TEXTLIST tlStations
  200 = 'Loading Station' | EN: 'Loading Station' | PL: 'Stacja Ladowania'
  201 = 'Weighing Station' | EN: 'Weighing Station' | PL: 'Stacja Wazenia'
  202 = 'Unloading Station' | EN: 'Unloading Station' | PL: 'Stacja Rozladowania'
   = ''
END_TEXTLIST

(* stored: Version 1.1.0.1, ProductVersion 3.1.4024.16
   TextList tlStations: Id {f51dacd5-1dfd-48d5-b111-c8439fb2fa2b} *)
